# EPICS substitutions: evrSupport/Db/ioc/IOC-LI21-PM01pattern.substitutions
#
# Pattern records
file evrPatternAll.db {
#	    Device        ,  SLC Pattern Check LNK    , EVR/Trigger
#	                                                  Links
  pattern { DEVICE        ,        LINK4              , LINK5 , LINK6 , TREF }
	  { IOC:LI21:PM01 ,         ""                ,  ""   ,  ""   , 1.03E06 }
}
file evrEventAll.db {
  pattern { DEVICE        }
	  { IOC:LI21:PM01 }
}
